TYPE ST_PowerControl_PsTarget_Measurements :
STRUCT
	r_PhaseVoltage					: REAL;
	r_ActivePower					: REAL;
	r_ReactivePower					: REAL;
END_STRUCT
END_TYPE

(* stored: Version 1.1.0.1, ProductVersion 3.1.4026.18
   DUT ST_PowerControl_PsTarget_Measurements: Id {afee19f6-e15c-4c4f-a1e1-6350848fab6e} *)
